Staubli VAL3: interpolateJ.pgx

public program interpolateJ(joint p_j1, joint p_j2, num p_nInterpolate, joint& x_jRetVal[], bool& x_bRetVal[])
begin
  // Interpolierten Jointwert berechnen
  x_jRetVal.j1=(p_j2.j1-p_j1.j1)*p_nInterpolate+p_j1.j1
  x_jRetVal.j2=(p_j2.j2-p_j1.j2)*p_nInterpolate+p_j1.j2
  x_jRetVal.j3=(p_j2.j3-p_j1.j3)*p_nInterpolate+p_j1.j3
  x_jRetVal.j4=(p_j2.j4-p_j1.j4)*p_nInterpolate+p_j1.j4
  x_jRetVal.j5=(p_j2.j5-p_j1.j5)*p_nInterpolate+p_j1.j5
  x_jRetVal.j6=(p_j2.j6-p_j1.j6)*p_nInterpolate+p_j1.j6
  x_bRetVal=isInRange(x_jRetVal)
end
